(* CODESYS project INDEX.project

Project tree, tasks and I/O mapping:
  Device : CODESYS Control Win V3, 3S - Smart Software Solutions GmbH, order no. 305021, version 3.5.11.30
    application Application
      libraries: Standard, * (System)
      task MainTask (cyclic, interval t#20ms, priority 1) calls PLC_PRG
      program PLC_PRG [FBD]
*)

// Device/Application/PLC_PRG
PROGRAM PLC_PRG
VAR
	S2: BOOL;
	P1: BOOL;
	S0: BOOL;
	S3: BOOL;
	P2: BOOL;
	P3: BOOL;
	CTU_1: CTU;
	CV1: WORD;
	P4: BOOL;
	TAP2: BOOL;
	TAP1: BOOL;
	A0: BOOL;
	A: BOOL;
	A1: BOOL;
	AVANCO: BOOL;
	RETORNO: BOOL;
END_VAR

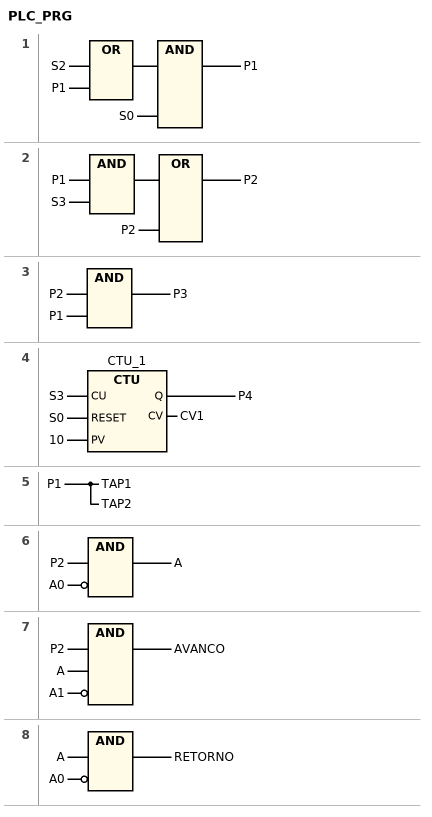
// NETWORK 1
P1 := (S2 OR P1) AND S0;

// NETWORK 2
P2 := P1 AND S3 OR P2;

// NETWORK 3
P3 := P2 AND P1;

// NETWORK 4
CTU_1(CU := S3, RESET := S0, PV := 10, CV => CV1); // CTU
P4 := CTU_1.Q;

// NETWORK 5
TAP1 := P1;
TAP2 := P1;

// NETWORK 6
A := P2 AND NOT A0;

// NETWORK 7
AVANCO := P2 AND A AND NOT A1;

// NETWORK 8
RETORNO := A AND NOT A0;

END_PROGRAM
